TYPE csp_transfer_upstacker_status_enum :
(
	CSP_TRANSFER_UPSTACKER_STATUS_NOT_INITIALIZED 							:=  0,
	CSP_TRANSFER_UPSTACKER_STATUS_DISABLED 									:=  10,
	CSP_TRANSFER_UPSTACKER_STATUS_ENABLE_REQUEST 							:=  20,
	CSP_TRANSFER_UPSTACKER_STATUS_ENABLING 									:=  30,
	CSP_TRANSFER_UPSTACKER_STATUS_ENABLED 									:=  40,
	CSP_TRANSFER_UPSTACKER_STATUS_HOME_REQUEST								:=  50,
	CSP_TRANSFER_UPSTACKER_STATUS_HOMING									:=  60,
	CSP_TRANSFER_UPSTACKER_STATUS_HOME_DONE									:=  70,
	CSP_TRANSFER_UPSTACKER_STATUS_CALCULATING_SLAVE_POSITION				:=  90,
	CSP_TRANSFER_UPSTACKER_STATUS_WAITING_SLAVE_ENGAGE						:= 100,
	CSP_TRANSFER_UPSTACKER_STATUS_PHASE_REQUEST								:= 140,
	CSP_TRANSFER_UPSTACKER_STATUS_PHASING									:= 150,
	CSP_TRANSFER_UPSTACKER_STATUS_PHASED									:= 160,
	CSP_TRANSFER_UPSTACKER_STATUS_CAM_ENGAGED_REQ							:= 170,
	CSP_TRANSFER_UPSTACKER_STATUS_AXIS_ENGAGE_VERIFY						:= 180,
	CSP_TRANSFER_UPSTACKER_STATUS_CAM_ON									:= 190,
	CSP_TRANSFER_UPSTACKER_STATUS_CAM_TABLE_READ							:= 195,
	CSP_TRANSFER_UPSTACKER_STATUS_CALCULATE_SLAVE_POSITION_REQUEST			:= 196,
	CSP_TRANSFER_UPSTACKER_STATUS_READY										:= 197,
	CSP_TRANSFER_UPSTACKER_STATUS_RUNNING_CAM								:= 200,
	CSP_TRANSFER_UPSTACKER_STATUS_CAM_OFF									:= 201,
	CSP_TRANSFER_UPSTACKER_STATUS_MOVING									:= 205,
	CSP_TRANSFER_UPSTACKER_STATUS_DISENGAGE									:= 210,
	CSP_TRANSFER_UPSTACKER_STATUS_DISENGAGING								:= 211,	
	CSP_TRANSFER_UPSTACKER_STATUS_STOP_REQUEST 								:= 500,
	CSP_TRANSFER_UPSTACKER_STATUS_DISABLE_REQUEST 							:= 530,
	CSP_TRANSFER_UPSTACKER_STATUS_DISABLING 								:= 540
) := CSP_TRANSFER_UPSTACKER_STATUS_NOT_INITIALIZED;
END_TYPE

(* stored: Version 1.1.0.1, ProductVersion 3.1.4022.12
   DUT csp_transfer_upstacker_status_enum: Id {40f884af-3d5b-4cde-a0ab-584711f61a22} *)
